(* Logix 5000 project; controller VET 1756-L62 rev 19.52; software revision 19.01; part 21 of 27 *)
(* tags used below, declared in another part *)
   _reset_locales : DINT;
   Batch : batch[10];
   Batch_buff : batch;
   Batch_Reportes : batch[100];
   comandos : DINT[10];
   db_input_cola : cola_almacenes;
   db_input_cola_batch_res : DINT;
   db_input_cola_flag : BOOL;
   dosificador : dosif_struct[20];
   Dosificar_LIQ_01 : PHASE;
   Dosificar_MAC_01 : PHASE;
   Dosificar_MAN_01 : PHASE;
   Dosificar_MIC_01 : PHASE;
   Dosificar_MIC_02 : PHASE;
   Dosificar_MID_01 : PHASE;
   hora_plc : DINT;
(* Interfaz_Equipment_Phase, continued *)

ROUTINE Dosificar_MIC_02   (* ladder *)
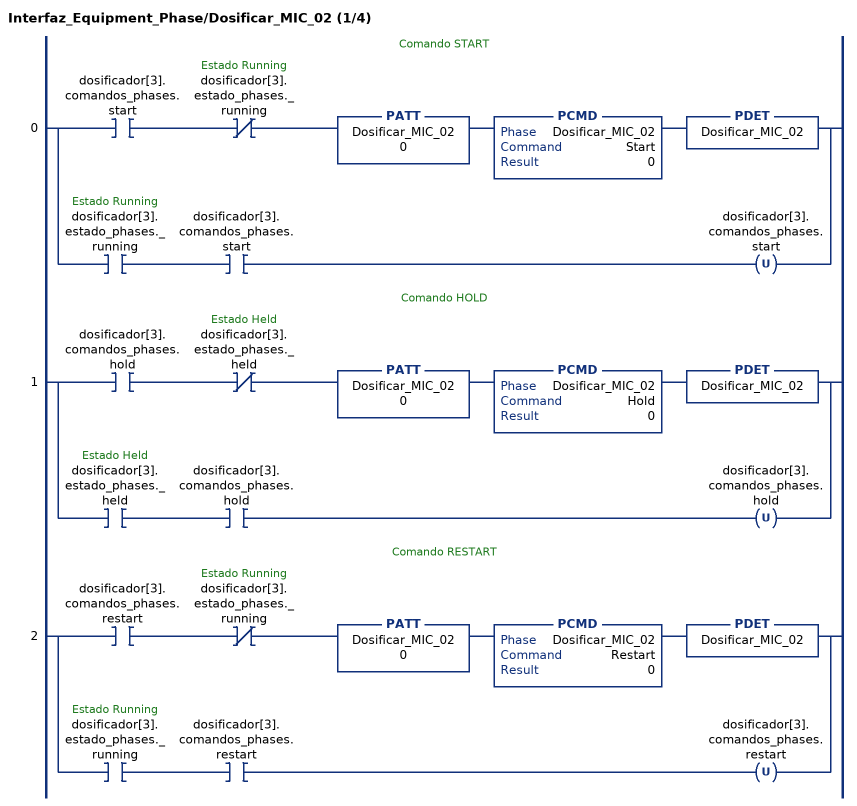
   // Comando START
   0: [XIC(dosificador[3].comandos_phases.start) XIO(dosificador[3].estado_phases._running) PATT(Dosificar_MIC_02,0) PCMD(Dosificar_MIC_02,Start,0) PDET(Dosificar_MIC_02) ,XIC(dosificador[3].estado_phases._running) XIC(dosificador[3].comandos_phases.start) OTU(dosificador[3].comandos_phases.start) ];
   // Comando HOLD
   1: [XIC(dosificador[3].comandos_phases.hold) XIO(dosificador[3].estado_phases._held) PATT(Dosificar_MIC_02,0) PCMD(Dosificar_MIC_02,Hold,0) PDET(Dosificar_MIC_02) ,XIC(dosificador[3].estado_phases._held) XIC(dosificador[3].comandos_phases.hold) OTU(dosificador[3].comandos_phases.hold) ];
   // Comando RESTART
   2: [XIC(dosificador[3].comandos_phases.restart) XIO(dosificador[3].estado_phases._running) PATT(Dosificar_MIC_02,0) PCMD(Dosificar_MIC_02,Restart,0) PDET(Dosificar_MIC_02) ,XIC(dosificador[3].estado_phases._running) XIC(dosificador[3].comandos_phases.restart) OTU(dosificador[3].comandos_phases.restart) ];
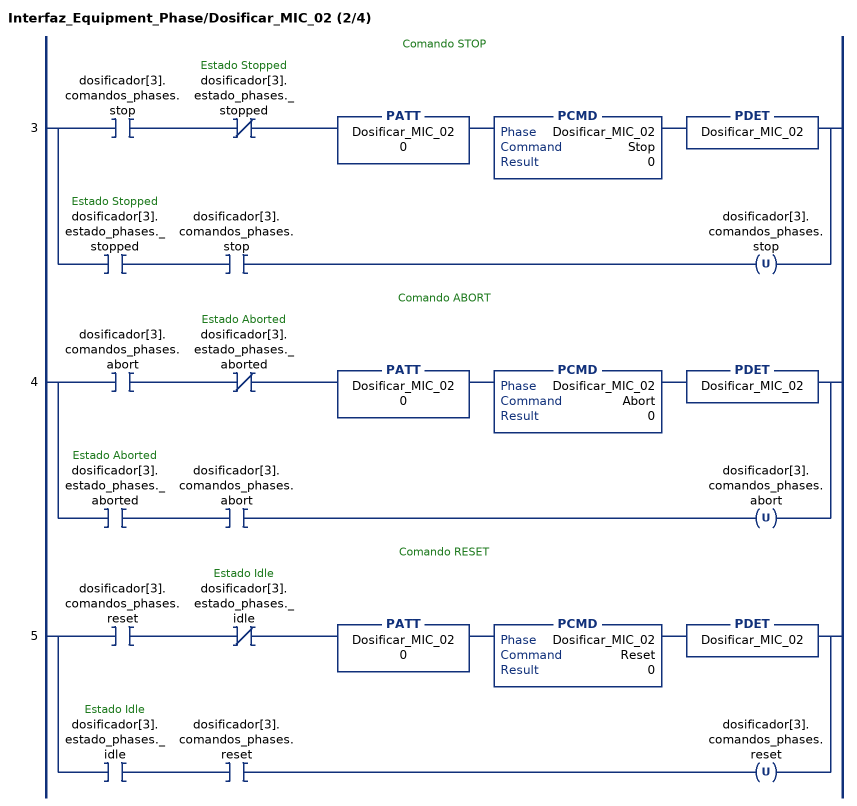
   // Comando STOP
   3: [XIC(dosificador[3].comandos_phases.stop) XIO(dosificador[3].estado_phases._stopped) PATT(Dosificar_MIC_02,0) PCMD(Dosificar_MIC_02,Stop,0) PDET(Dosificar_MIC_02) ,XIC(dosificador[3].estado_phases._stopped) XIC(dosificador[3].comandos_phases.stop) OTU(dosificador[3].comandos_phases.stop) ];
   // Comando ABORT
   4: [XIC(dosificador[3].comandos_phases.abort) XIO(dosificador[3].estado_phases._aborted) PATT(Dosificar_MIC_02,0) PCMD(Dosificar_MIC_02,Abort,0) PDET(Dosificar_MIC_02) ,XIC(dosificador[3].estado_phases._aborted) XIC(dosificador[3].comandos_phases.abort) OTU(dosificador[3].comandos_phases.abort) ];
   // Comando RESET
   5: [XIC(dosificador[3].comandos_phases.reset) XIO(dosificador[3].estado_phases._idle) PATT(Dosificar_MIC_02,0) PCMD(Dosificar_MIC_02,Reset,0) PDET(Dosificar_MIC_02) ,XIC(dosificador[3].estado_phases._idle) XIC(dosificador[3].comandos_phases.reset) OTU(dosificador[3].comandos_phases.reset) ];
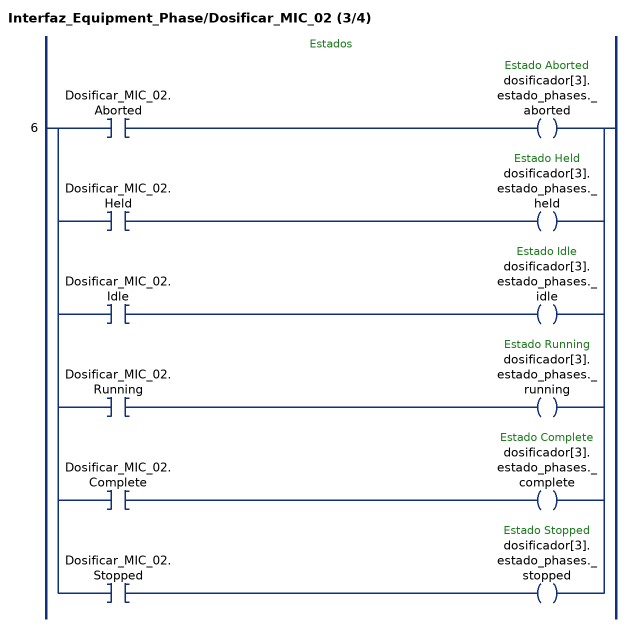
   // Estados
   6: [XIC(Dosificar_MIC_02.Aborted) OTE(dosificador[3].estado_phases._aborted) ,XIC(Dosificar_MIC_02.Held) OTE(dosificador[3].estado_phases._held) ,XIC(Dosificar_MIC_02.Idle) OTE(dosificador[3].estado_phases._idle) ,XIC(Dosificar_MIC_02.Running) OTE(dosificador[3].estado_phases._running) ,XIC(Dosificar_MIC_02.Complete) OTE(dosificador[3].estado_phases._complete) ,XIC(Dosificar_MIC_02.Stopped) OTE(dosificador[3].estado_phases._stopped) ];
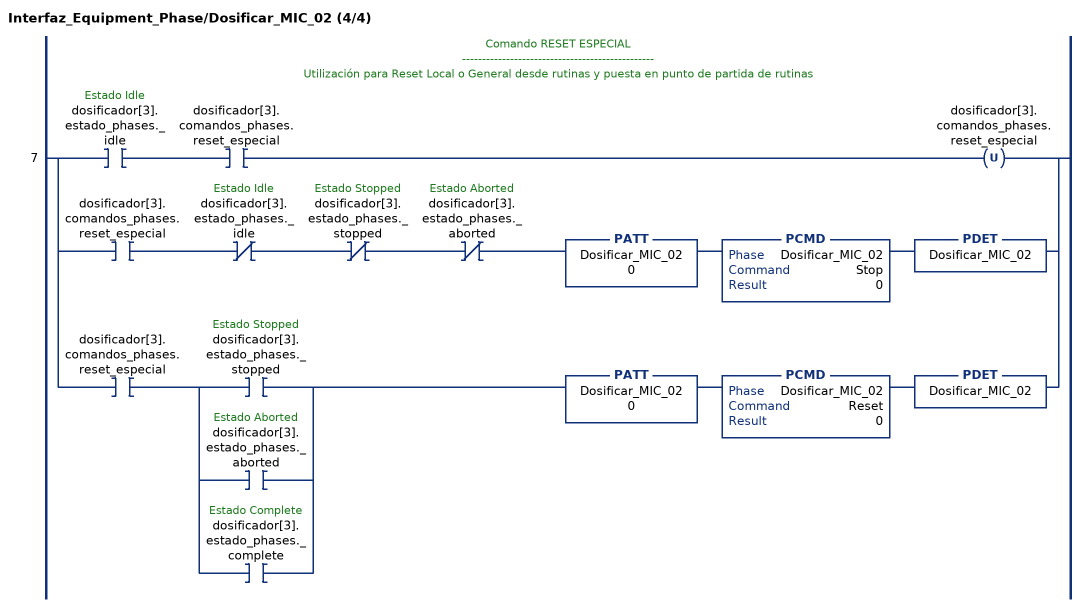
   // Comando RESET ESPECIAL
   // ------------------------------------------------
   // Utilización para Reset Local o General desde rutinas y puesta en punto de partida de rutinas
   7: [XIC(dosificador[3].estado_phases._idle) XIC(dosificador[3].comandos_phases.reset_especial) OTU(dosificador[3].comandos_phases.reset_especial) ,XIC(dosificador[3].comandos_phases.reset_especial) XIO(dosificador[3].estado_phases._idle) XIO(dosificador[3].estado_phases._stopped) XIO(dosificador[3].estado_phases._aborted) PATT(Dosificar_MIC_02,0) PCMD(Dosificar_MIC_02,Stop,0) PDET(Dosificar_MIC_02) ,XIC(dosificador[3].comandos_phases.reset_especial) [XIC(dosificador[3].estado_phases._stopped) ,XIC(dosificador[3].estado_phases._aborted) ,XIC(dosificador[3].estado_phases._complete) ] PATT(Dosificar_MIC_02,0) PCMD(Dosificar_MIC_02,Reset,0) PDET(Dosificar_MIC_02) ];
END_ROUTINE

ROUTINE Dosificar_MID_01   (* ladder *)
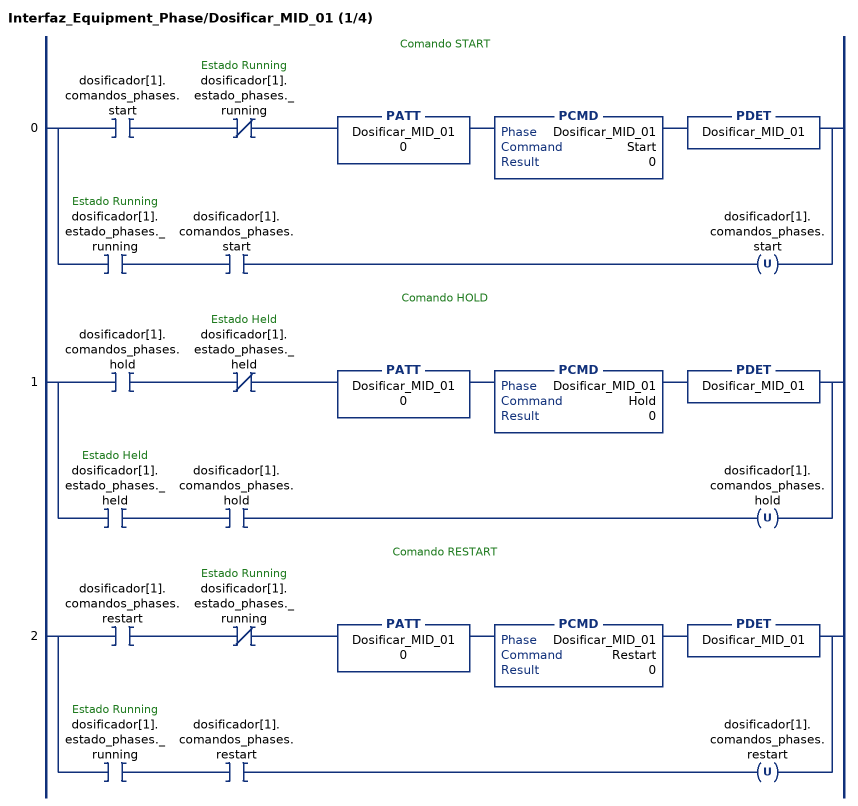
   // Comando START
   0: [XIC(dosificador[1].comandos_phases.start) XIO(dosificador[1].estado_phases._running) PATT(Dosificar_MID_01,0) PCMD(Dosificar_MID_01,Start,0) PDET(Dosificar_MID_01) ,XIC(dosificador[1].estado_phases._running) XIC(dosificador[1].comandos_phases.start) OTU(dosificador[1].comandos_phases.start) ];
   // Comando HOLD
   1: [XIC(dosificador[1].comandos_phases.hold) XIO(dosificador[1].estado_phases._held) PATT(Dosificar_MID_01,0) PCMD(Dosificar_MID_01,Hold,0) PDET(Dosificar_MID_01) ,XIC(dosificador[1].estado_phases._held) XIC(dosificador[1].comandos_phases.hold) OTU(dosificador[1].comandos_phases.hold) ];
   // Comando RESTART
   2: [XIC(dosificador[1].comandos_phases.restart) XIO(dosificador[1].estado_phases._running) PATT(Dosificar_MID_01,0) PCMD(Dosificar_MID_01,Restart,0) PDET(Dosificar_MID_01) ,XIC(dosificador[1].estado_phases._running) XIC(dosificador[1].comandos_phases.restart) OTU(dosificador[1].comandos_phases.restart) ];
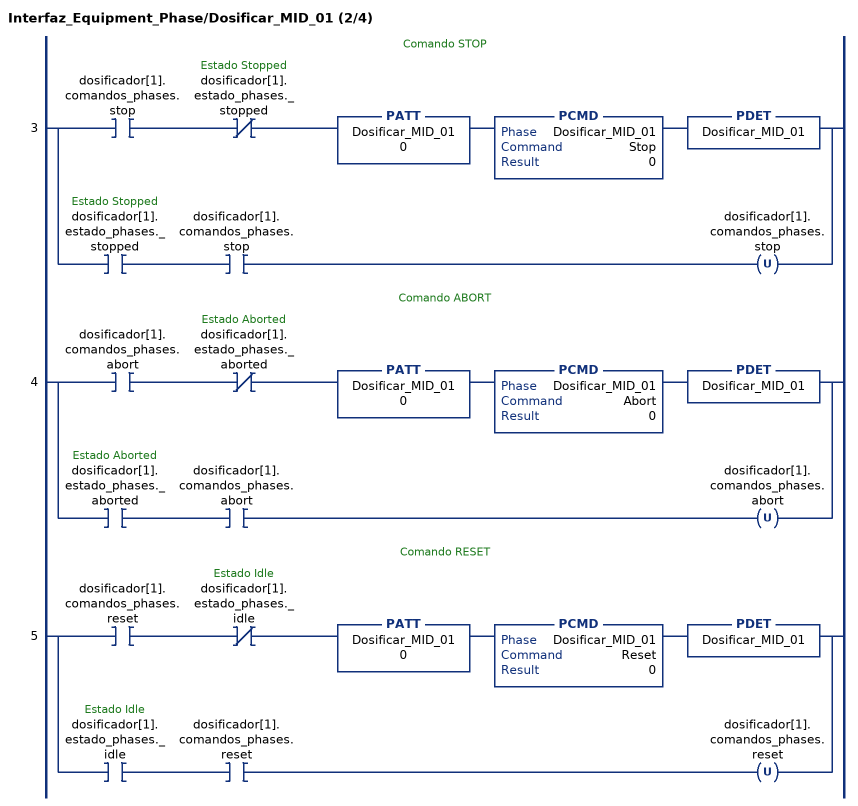
   // Comando STOP
   3: [XIC(dosificador[1].comandos_phases.stop) XIO(dosificador[1].estado_phases._stopped) PATT(Dosificar_MID_01,0) PCMD(Dosificar_MID_01,Stop,0) PDET(Dosificar_MID_01) ,XIC(dosificador[1].estado_phases._stopped) XIC(dosificador[1].comandos_phases.stop) OTU(dosificador[1].comandos_phases.stop) ];
   // Comando ABORT
   4: [XIC(dosificador[1].comandos_phases.abort) XIO(dosificador[1].estado_phases._aborted) PATT(Dosificar_MID_01,0) PCMD(Dosificar_MID_01,Abort,0) PDET(Dosificar_MID_01) ,XIC(dosificador[1].estado_phases._aborted) XIC(dosificador[1].comandos_phases.abort) OTU(dosificador[1].comandos_phases.abort) ];
   // Comando RESET
   5: [XIC(dosificador[1].comandos_phases.reset) XIO(dosificador[1].estado_phases._idle) PATT(Dosificar_MID_01,0) PCMD(Dosificar_MID_01,Reset,0) PDET(Dosificar_MID_01) ,XIC(dosificador[1].estado_phases._idle) XIC(dosificador[1].comandos_phases.reset) OTU(dosificador[1].comandos_phases.reset) ];
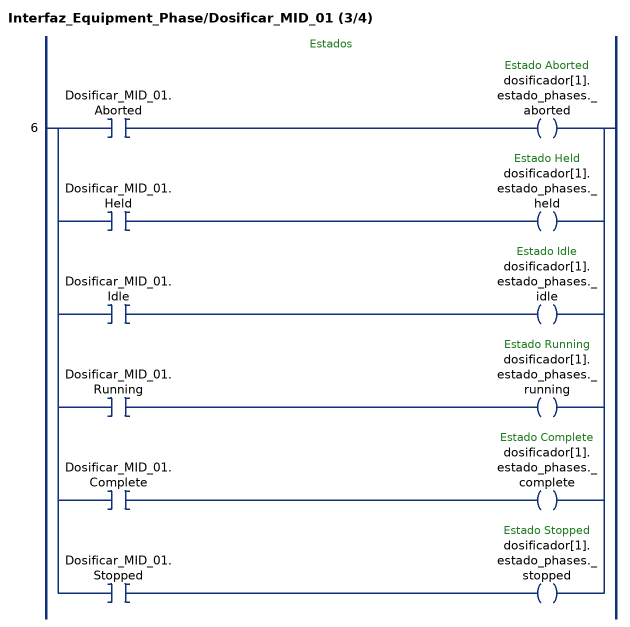
   // Estados
   6: [XIC(Dosificar_MID_01.Aborted) OTE(dosificador[1].estado_phases._aborted) ,XIC(Dosificar_MID_01.Held) OTE(dosificador[1].estado_phases._held) ,XIC(Dosificar_MID_01.Idle) OTE(dosificador[1].estado_phases._idle) ,XIC(Dosificar_MID_01.Running) OTE(dosificador[1].estado_phases._running) ,XIC(Dosificar_MID_01.Complete) OTE(dosificador[1].estado_phases._complete) ,XIC(Dosificar_MID_01.Stopped) OTE(dosificador[1].estado_phases._stopped) ];
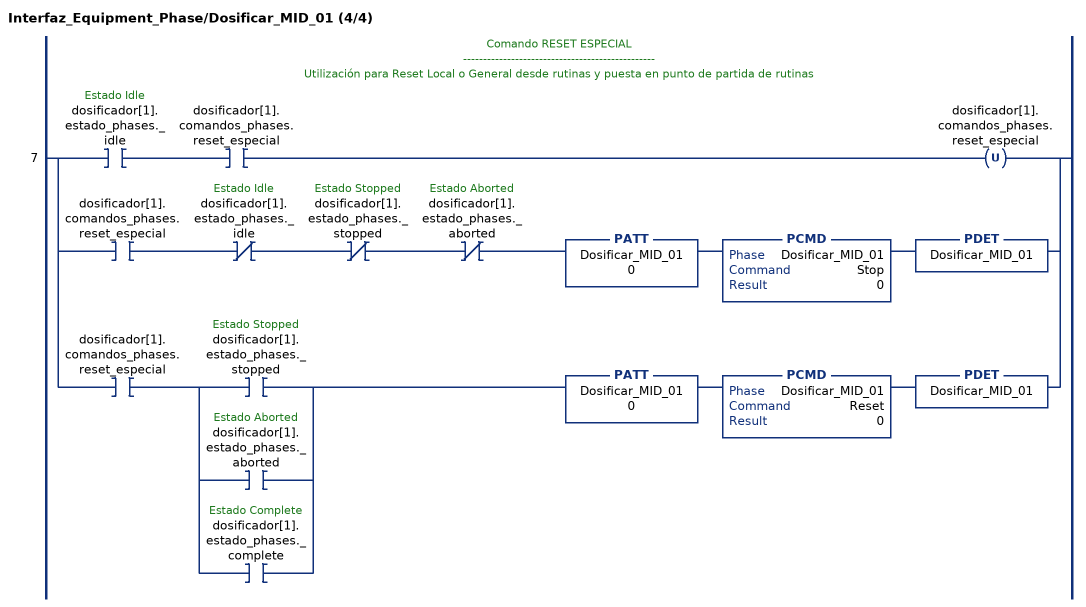
   // Comando RESET ESPECIAL
   // ------------------------------------------------
   // Utilización para Reset Local o General desde rutinas y puesta en punto de partida de rutinas
   7: [XIC(dosificador[1].estado_phases._idle) XIC(dosificador[1].comandos_phases.reset_especial) OTU(dosificador[1].comandos_phases.reset_especial) ,XIC(dosificador[1].comandos_phases.reset_especial) XIO(dosificador[1].estado_phases._idle) XIO(dosificador[1].estado_phases._stopped) XIO(dosificador[1].estado_phases._aborted) PATT(Dosificar_MID_01,0) PCMD(Dosificar_MID_01,Stop,0) PDET(Dosificar_MID_01) ,XIC(dosificador[1].comandos_phases.reset_especial) [XIC(dosificador[1].estado_phases._stopped) ,XIC(dosificador[1].estado_phases._aborted) ,XIC(dosificador[1].estado_phases._complete) ] PATT(Dosificar_MID_01,0) PCMD(Dosificar_MID_01,Reset,0) PDET(Dosificar_MID_01) ];
END_ROUTINE

ROUTINE main   (* ladder *)
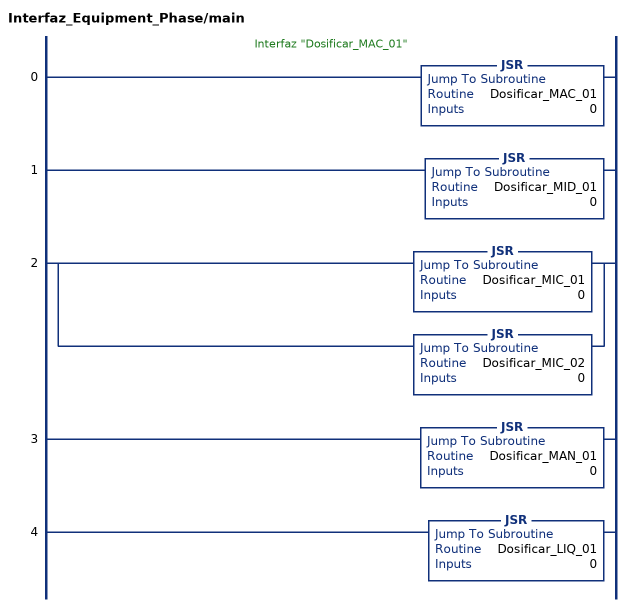
   // Interfaz "Dosificar_MAC_01"
   0: JSR(Dosificar_MAC_01,0);
   1: JSR(Dosificar_MID_01,0);
   2: [JSR(Dosificar_MIC_01,0) ,JSR(Dosificar_MIC_02,0) ];
   3: JSR(Dosificar_MAN_01,0);
   4: JSR(Dosificar_LIQ_01,0);
END_ROUTINE
END_PROGRAM

PROGRAM Main   (* main routine main *)
VAR
   _reset_local : ALIAS FOR _reset_locales.0;
   batch_in : batch := (Head.folio := 32, Head.orden := -3, Head.formula := 'DUMMY', Head.estado := 5, Head.correlativo := 2, Head.total_batch := 20, Head.peso_teorico := 1733.0, Data.codigo[0] := 81, Data.codigo[1] := 51, Data.codigo[2] := 53, Data.codigo[3] := 55, Data.codigo[4] := 57, Data.codigo[5] := 67, Data.codigo[6] := 68, Data.codigo[7] := 69, Data.codigo[8] := 70, Data.codigo[9] := 74, Data.codigo[10] := 75, Data.codigo[11] := 76, Data.codigo[12] := 77, Data.codigo[13] := 60, Data.codigo[14] := 62, Data.codigo[15] := 64, Data.codigo[16] := 66, Data.peso_f[0] := 70.0, Data.peso_f[1] := 400.0, Data.peso_f[2] := 350.0, Data.peso_f[3] := 175.0, Data.peso_f[4] := 225.0, Data.peso_f[5] := 30.0, Data.peso_f[6] := 25.0, Data.peso_f[7] := 17.5, Data.peso_f[8] := 17.5, Data.peso_f[9] := 30.0, Data.peso_f[10] := 5.0, Data.peso_f[11] := 4.0, Data.peso_f[12] := 4.0, Data.peso_f[13] := 125.0, Data.peso_f[14] := 125.0, Data.peso_f[15] := 65.0, Data.peso_f[16] := 65.0);
   batch_out : batch;
   db1_var_batch : variables_procedimientos := (trigger[0] := 1, trigger[1] := 1, trigger[2] := 1, trigger[3] := 1, handshake[0] := 1, handshake[1] := 1, handshake[2] := 1, in_tstamp[0] := 18273253, in_tstamp[1] := 18273653, in_tstamp[2] := 18274003, in_tstamp[3] := 11123107, out_tstamp[0] := 18273253, out_tstamp[2] := 18274003, D[0] := 3, D[1] := 32, T[0].PRE := 2000, T[1].PRE := 10000, T[2].PRE := 2000, T[3].PRE := 10000, T[4].PRE := 2000, T[5].PRE := 10000);
        .D[0].1   // Habilitación Recepción Automática
        .D[0].0   // Resumen Dehabilitación
        .D[0]   // Bits Estados
        .D[1]   // Folio - Pedir batch
   db2_cola_res : DINT[20] := ([0] := 32, [1] := 27862, [2] := 39951);
   db2_var_res : variables_procedimientos := (step_idx := 20, trigger[0] := 1, handshake[0] := -1, in_tstamp[0] := 18464153, D[0] := 32, i0 := 1, SetD[0] := 20, T[0].PRE := 3000, T[1].PRE := 10000, T[1].ACC := 4992, T[1].EN := 1, T[1].TT := 1);
   db3_var_rep : variables_procedimientos;
   db4_cola_mc : cola_almacenes[100] := ([0].origen := 31, [0].destino := 1000, [0].cantidad := 16.200012, [0].folio_op := 39951, [0].fecha := 20140306, [0].hora := 1163858, [1].origen := 31, [1].destino := 1000, [1].cantidad := 16.299988, [1].folio_op := 39973, [1].fecha := 20140306, [1].hora := 1170439, [2].origen := 71, [2].destino := 1000, [2].cantidad := 2.015625, [2].folio_op := 39973, [2].fecha := 20140306, [2].hora := 1170440, [3].origen := 31, [3].destino := 1000, [3].cantidad := 16.600006, [3].folio_op := 39975, [3].fecha := 20140306, [3].hora := 1172638, [4].origen := 70, [4].destino := 1000, [4].cantidad := 31.046875, [4].folio_op := 39889, [4].fecha := 20140306, [4].hora := 1174046, [5].origen := 31, [5].destino := 1000, [5].cantidad := 16.800018, [5].folio_op := 39977, [5].fecha := 20140306, [5].hora := 1175226, [6].origen := 32, [6].destino := 1000, [6].cantidad := 10.300018, [6].folio_op := 39977, [6].fecha := 20140306, [6].hora := 1175710, [7].origen := 70, [7].destino := 1000, [7].cantidad := 31.0, [7].folio_op := 39815, [7].fecha := 20140306, [7].hora := 1122359, [8].origen := 71, [8].destino := 1000, [8].cantidad := 2.0, [8].folio_op := 39937, [8].fecha := 20140306, [8].hora := 1124946, [9].origen := 31, [9].destino := 1000, [9].cantidad := 16.800018, [9].folio_op := 39937, [9].fecha := 20140306, [9].hora := 1124947,
        [10].origen := 19, [10].destino := 1000, [10].cantidad := 656.0, [10].folio_op := 39903, [10].fecha := 20140306, [10].hora := 1125834, [11].origen := 31, [11].destino := 1000, [11].cantidad := 16.299988, [11].folio_op := 39942, [11].fecha := 20140306, [11].hora := 1135834, [12].origen := 101, [12].destino := 1000, [12].cantidad := 50.4375, [12].folio_op := 39904, [12].fecha := 20140306, [12].hora := 1141004, [13].origen := 16, [13].destino := 25, [14].origen := 16, [14].destino := 25, [15].origen := 31, [15].destino := 1000, [15].cantidad := 16.5, [15].folio_op := 39945, [15].fecha := 20140306, [15].hora := 1151258, [16].origen := 31, [16].destino := 1000, [16].cantidad := 16.5, [16].folio_op := 39946, [16].fecha := 20140306, [16].hora := 1152347, [17].origen := 31, [17].destino := 1000, [17].cantidad := 16.799988, [17].folio_op := 39947, [17].fecha := 20140306, [17].hora := 1153707, [18].origen := 31, [18].destino := 1000, [18].cantidad := 16.200012, [18].folio_op := 39948, [18].fecha := 20140306, [18].hora := 1160218, [19].origen := 31, [19].destino := 1000, [19].cantidad := 16.800003, [19].folio_op := 39949, [19].fecha := 20140306, [19].hora := 1161219);
   db4_var_mc : variables_procedimientos;
   db5_var_rep : variables_procedimientos := (i0 := 50, i1 := 50, SetD[0] := 100);
        .I0   // Largo Actual Cola
        .SETD[0]   // Largo Maximo Cola
        .I1   // Próximo a la Cola
        .I2   // Primero en Cola
   var_wd : variables_procedimientos := (step_idx := 10, in_tstamp[0] := 18464753, T[0].PRE := 20000, T[0].ACC := 1992, T[0].EN := 1, T[0].TT := 1, T[1].PRE := 10000);
   watchdog : BOOL;
END_VAR

ROUTINE aux_manejo_cola   (* ladder *)
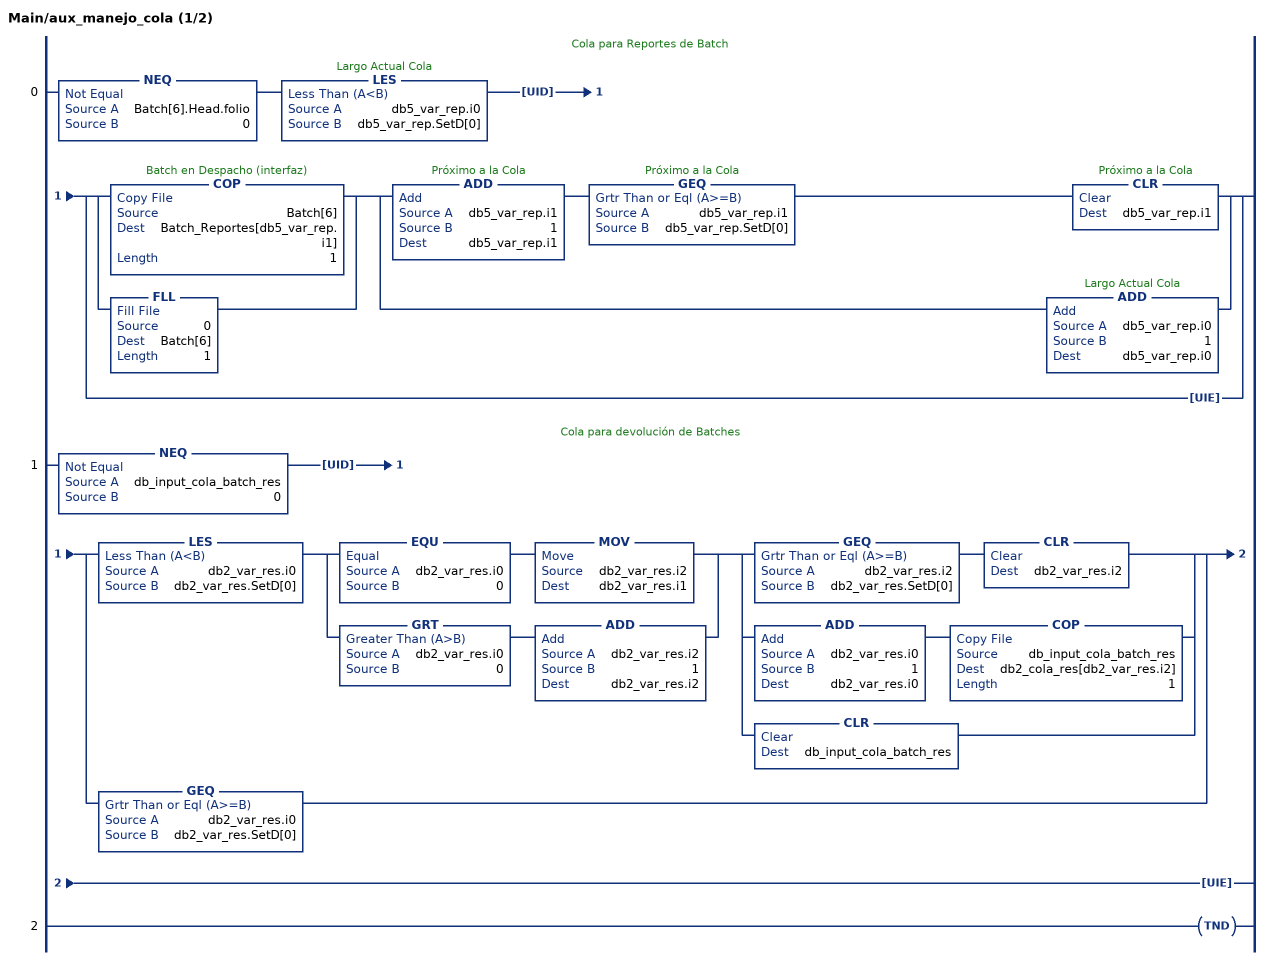
   // Cola para Reportes de Batch
   0: NEQ(Batch[6].Head.folio,0)LES(db5_var_rep.i0,db5_var_rep.SetD[0])UID()[[COP(Batch[6],Batch_Reportes[db5_var_rep.i1],1) ,FLL(0,Batch[6],1) ] [ADD(db5_var_rep.i1,1,db5_var_rep.i1) GEQ(db5_var_rep.i1,db5_var_rep.SetD[0]) CLR(db5_var_rep.i1) ,ADD(db5_var_rep.i0,1,db5_var_rep.i0) ] ,UIE() ];
   // Cola para devolución de Batches
   1: NEQ(db_input_cola_batch_res,0)UID()[LES(db2_var_res.i0,db2_var_res.SetD[0]) [EQU(db2_var_res.i0,0) MOV(db2_var_res.i2,db2_var_res.i1) ,GRT(db2_var_res.i0,0) ADD(db2_var_res.i2,1,db2_var_res.i2) ] [GEQ(db2_var_res.i2,db2_var_res.SetD[0]) CLR(db2_var_res.i2) ,ADD(db2_var_res.i0,1,db2_var_res.i0) COP(db_input_cola_batch_res,db2_cola_res[db2_var_res.i2],1) ,CLR(db_input_cola_batch_res) ] ,GEQ(db2_var_res.i0,db2_var_res.SetD[0]) ]UIE();
   2: TND();
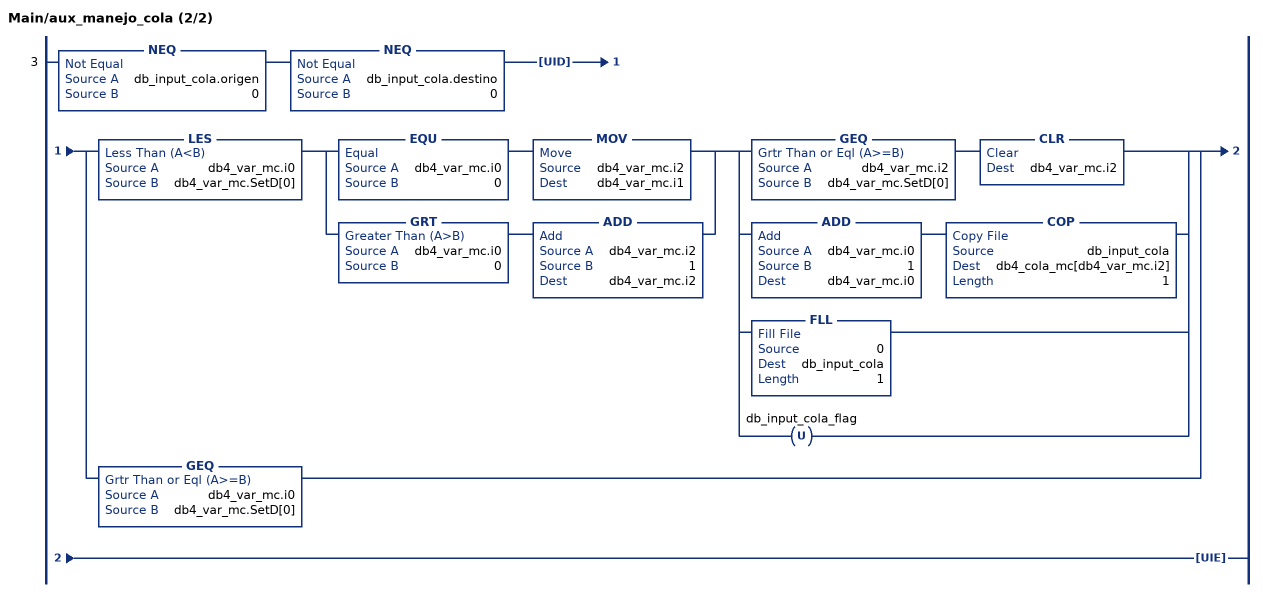
   3: NEQ(db_input_cola.origen,0)NEQ(db_input_cola.destino,0)UID()[LES(db4_var_mc.i0,db4_var_mc.SetD[0]) [EQU(db4_var_mc.i0,0) MOV(db4_var_mc.i2,db4_var_mc.i1) ,GRT(db4_var_mc.i0,0) ADD(db4_var_mc.i2,1,db4_var_mc.i2) ] [GEQ(db4_var_mc.i2,db4_var_mc.SetD[0]) CLR(db4_var_mc.i2) ,ADD(db4_var_mc.i0,1,db4_var_mc.i0) COP(db_input_cola,db4_cola_mc[db4_var_mc.i2],1) ,FLL(0,db_input_cola,1) ,OTU(db_input_cola_flag) ] ,GEQ(db4_var_mc.i0,db4_var_mc.SetD[0]) ]UIE();
END_ROUTINE

ROUTINE db0_watchdog   (* ladder *)
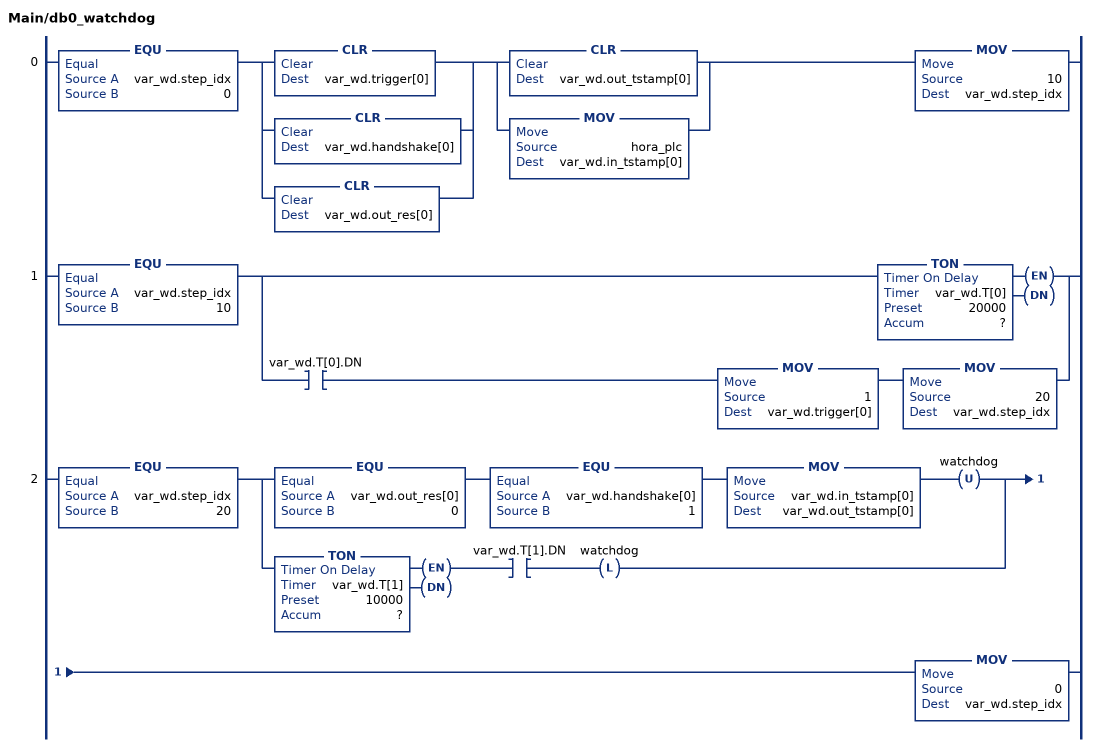
   0: EQU(var_wd.step_idx,0)[CLR(var_wd.trigger[0]) ,CLR(var_wd.handshake[0]) ,CLR(var_wd.out_res[0]) ][CLR(var_wd.out_tstamp[0]) ,MOV(hora_plc,var_wd.in_tstamp[0]) ]MOV(10,var_wd.step_idx);
   1: EQU(var_wd.step_idx,10)[TON(var_wd.T[0],?,?) ,XIC(var_wd.T[0].DN) MOV(1,var_wd.trigger[0]) MOV(20,var_wd.step_idx) ];
   2: EQU(var_wd.step_idx,20)[EQU(var_wd.out_res[0],0) EQU(var_wd.handshake[0],1) MOV(var_wd.in_tstamp[0],var_wd.out_tstamp[0]) OTU(watchdog) ,TON(var_wd.T[1],?,?) XIC(var_wd.T[1].DN) OTL(watchdog) ]MOV(0,var_wd.step_idx);
END_ROUTINE

ROUTINE db1_obtener_batch   (* ladder *)
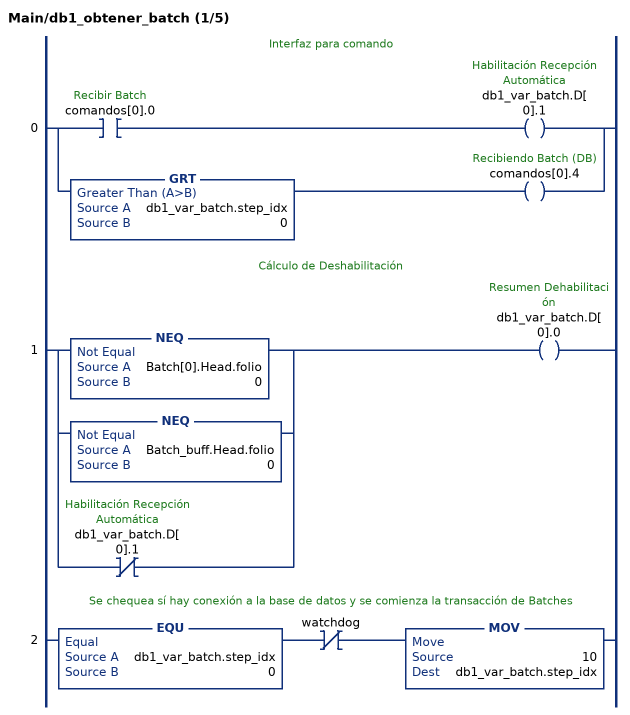
   // Interfaz para comando
   0: [XIC(comandos[0].0) OTE(db1_var_batch.D[0].1) ,GRT(db1_var_batch.step_idx,0) OTE(comandos[0].4) ];
   // Cálculo de Deshabilitación
   1: [NEQ(Batch[0].Head.folio,0) ,NEQ(Batch_buff.Head.folio,0) ,XIO(db1_var_batch.D[0].1) ]OTE(db1_var_batch.D[0].0);
   // Se chequea sí hay conexión a la base de datos y se comienza la transacción de Batches
   2: EQU(db1_var_batch.step_idx,0)XIO(watchdog)MOV(10,db1_var_batch.step_idx);
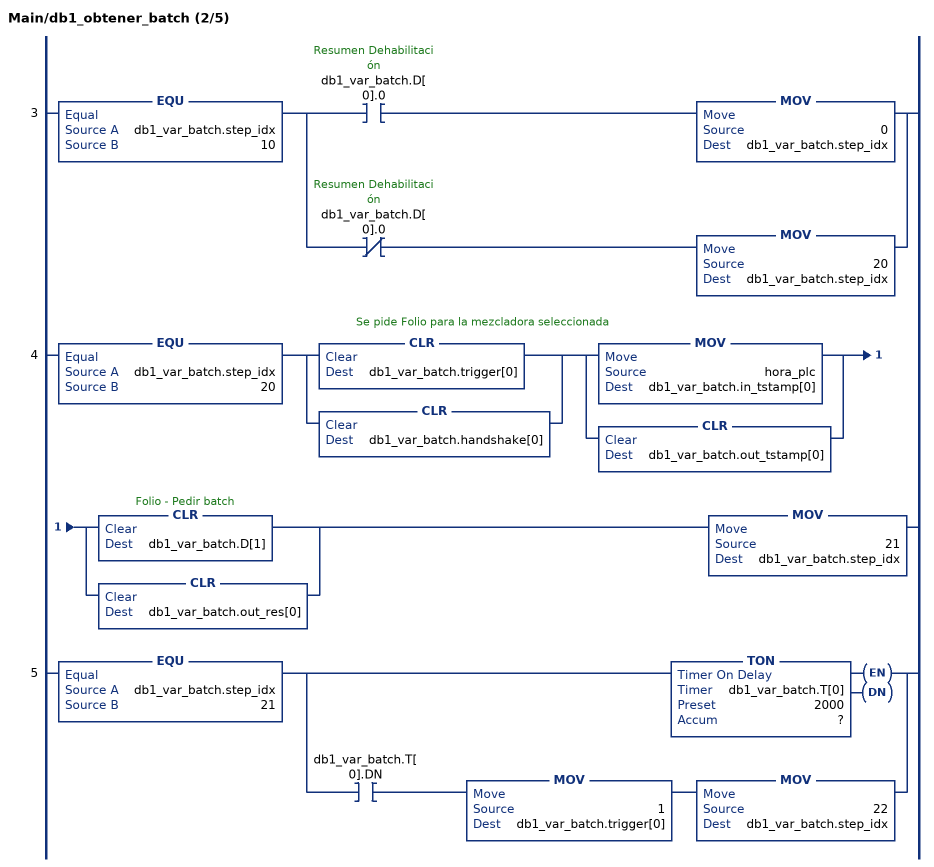
   3: EQU(db1_var_batch.step_idx,10)[XIC(db1_var_batch.D[0].0) MOV(0,db1_var_batch.step_idx) ,XIO(db1_var_batch.D[0].0) MOV(20,db1_var_batch.step_idx) ];
   // Se pide Folio para la mezcladora seleccionada
   4: EQU(db1_var_batch.step_idx,20)[CLR(db1_var_batch.trigger[0]) ,CLR(db1_var_batch.handshake[0]) ][MOV(hora_plc,db1_var_batch.in_tstamp[0]) ,CLR(db1_var_batch.out_tstamp[0]) ][CLR(db1_var_batch.D[1]) ,CLR(db1_var_batch.out_res[0]) ]MOV(21,db1_var_batch.step_idx);
   5: EQU(db1_var_batch.step_idx,21)[TON(db1_var_batch.T[0],?,?) ,XIC(db1_var_batch.T[0].DN) MOV(1,db1_var_batch.trigger[0]) MOV(22,db1_var_batch.step_idx) ];
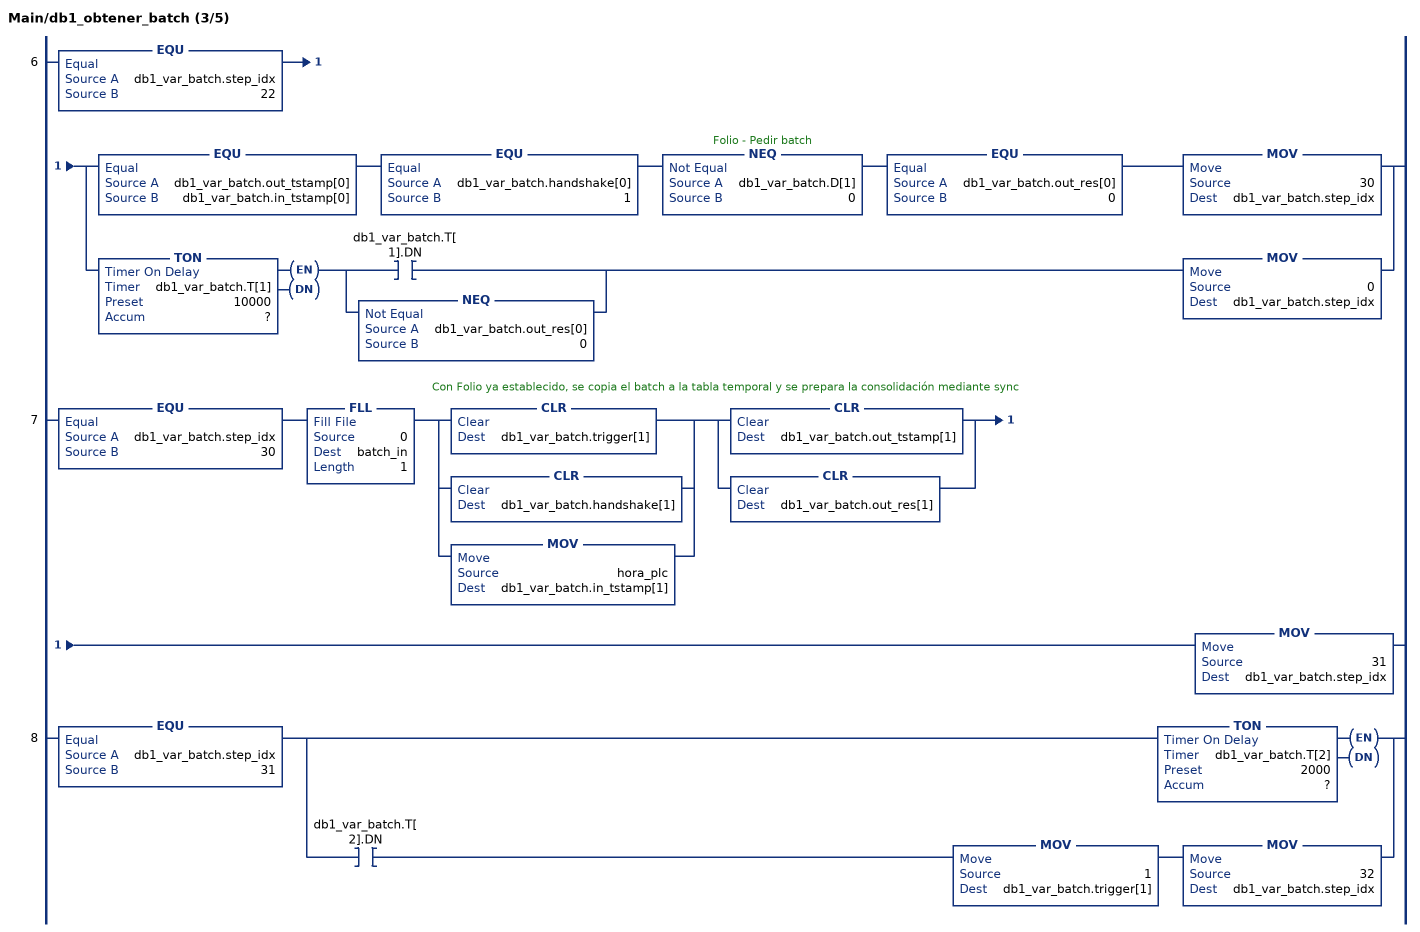
   6: EQU(db1_var_batch.step_idx,22)[EQU(db1_var_batch.out_tstamp[0],db1_var_batch.in_tstamp[0]) EQU(db1_var_batch.handshake[0],1) NEQ(db1_var_batch.D[1],0) EQU(db1_var_batch.out_res[0],0) MOV(30,db1_var_batch.step_idx) ,TON(db1_var_batch.T[1],?,?) [XIC(db1_var_batch.T[1].DN) ,NEQ(db1_var_batch.out_res[0],0) ] MOV(0,db1_var_batch.step_idx) ];
   // Con Folio ya establecido, se copia el batch a la tabla temporal y se prepara la consolidación mediante sync
   7: EQU(db1_var_batch.step_idx,30)FLL(0,batch_in,1)[CLR(db1_var_batch.trigger[1]) ,CLR(db1_var_batch.handshake[1]) ,MOV(hora_plc,db1_var_batch.in_tstamp[1]) ][CLR(db1_var_batch.out_tstamp[1]) ,CLR(db1_var_batch.out_res[1]) ]MOV(31,db1_var_batch.step_idx);
   8: EQU(db1_var_batch.step_idx,31)[TON(db1_var_batch.T[2],?,?) ,XIC(db1_var_batch.T[2].DN) MOV(1,db1_var_batch.trigger[1]) MOV(32,db1_var_batch.step_idx) ];
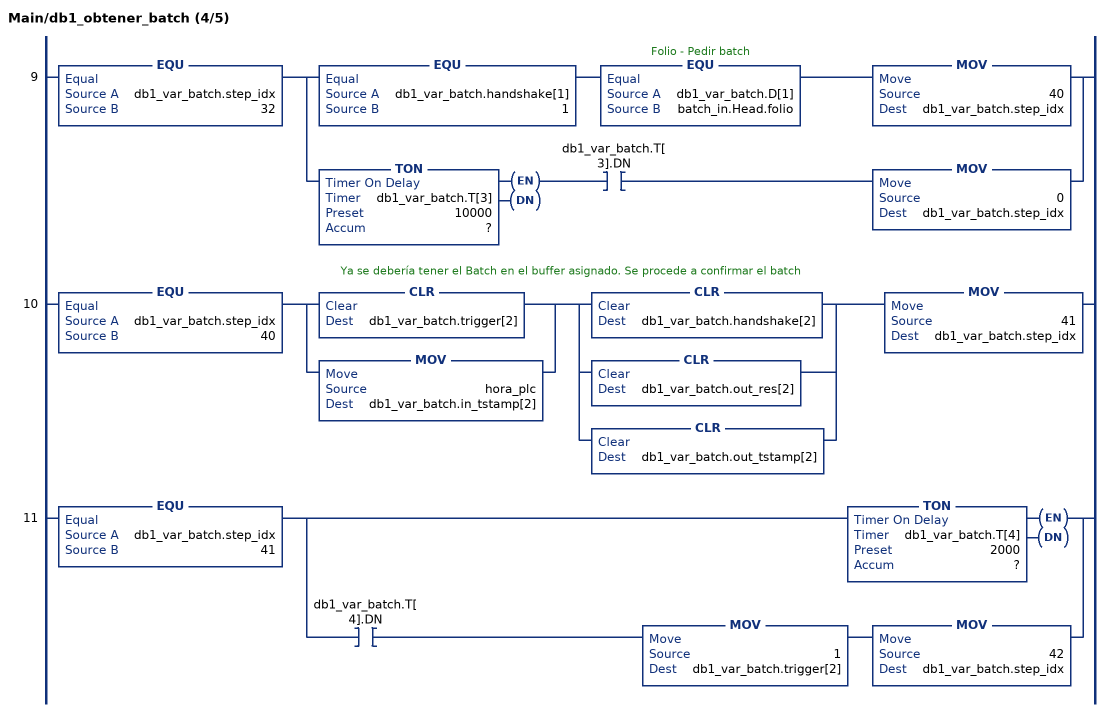
   9: EQU(db1_var_batch.step_idx,32)[EQU(db1_var_batch.handshake[1],1) EQU(db1_var_batch.D[1],batch_in.Head.folio) MOV(40,db1_var_batch.step_idx) ,TON(db1_var_batch.T[3],?,?) XIC(db1_var_batch.T[3].DN) MOV(0,db1_var_batch.step_idx) ];
   // Ya se debería tener el Batch en el buffer asignado. Se procede a confirmar el batch
   10: EQU(db1_var_batch.step_idx,40)[CLR(db1_var_batch.trigger[2]) ,MOV(hora_plc,db1_var_batch.in_tstamp[2]) ][CLR(db1_var_batch.handshake[2]) ,CLR(db1_var_batch.out_res[2]) ,CLR(db1_var_batch.out_tstamp[2]) ]MOV(41,db1_var_batch.step_idx);
   11: EQU(db1_var_batch.step_idx,41)[TON(db1_var_batch.T[4],?,?) ,XIC(db1_var_batch.T[4].DN) MOV(1,db1_var_batch.trigger[2]) MOV(42,db1_var_batch.step_idx) ];
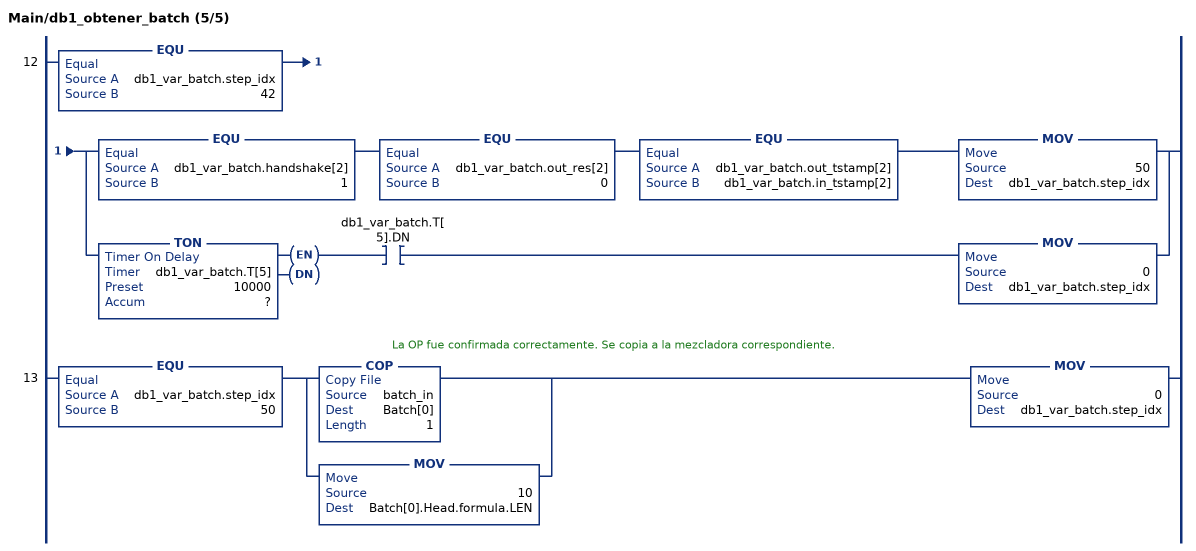
   12: EQU(db1_var_batch.step_idx,42)[EQU(db1_var_batch.handshake[2],1) EQU(db1_var_batch.out_res[2],0) EQU(db1_var_batch.out_tstamp[2],db1_var_batch.in_tstamp[2]) MOV(50,db1_var_batch.step_idx) ,TON(db1_var_batch.T[5],?,?) XIC(db1_var_batch.T[5].DN) MOV(0,db1_var_batch.step_idx) ];
   // La OP fue confirmada correctamente. Se copia a la mezcladora correspondiente.
   13: EQU(db1_var_batch.step_idx,50)[COP(batch_in,Batch[0],1) ,MOV(10,Batch[0].Head.formula.LEN) ]MOV(0,db1_var_batch.step_idx);
END_ROUTINE

ROUTINE db2_devolver_op   (* ladder *)
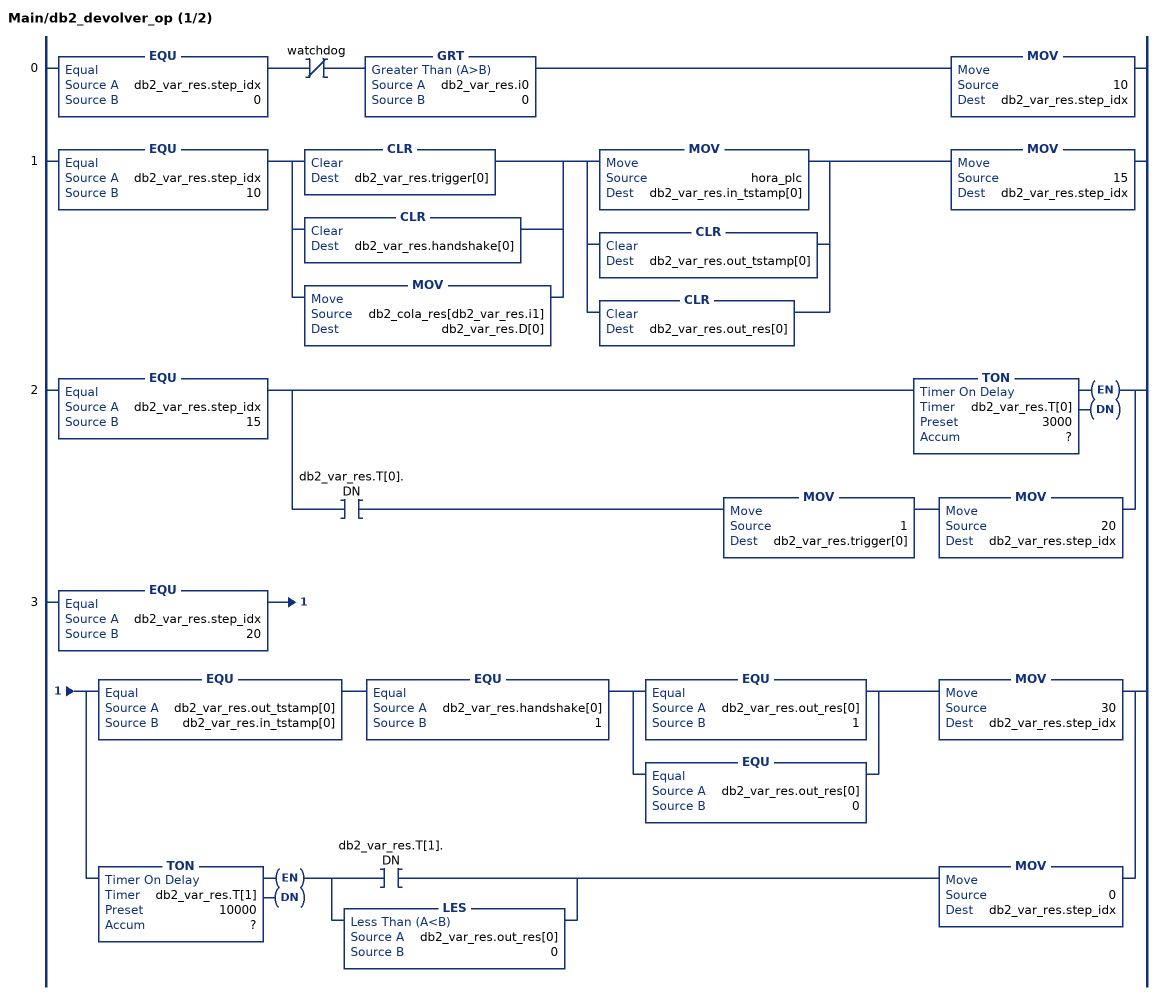
   0: EQU(db2_var_res.step_idx,0)XIO(watchdog)GRT(db2_var_res.i0,0)MOV(10,db2_var_res.step_idx);
   1: EQU(db2_var_res.step_idx,10)[CLR(db2_var_res.trigger[0]) ,CLR(db2_var_res.handshake[0]) ,MOV(db2_cola_res[db2_var_res.i1],db2_var_res.D[0]) ][MOV(hora_plc,db2_var_res.in_tstamp[0]) ,CLR(db2_var_res.out_tstamp[0]) ,CLR(db2_var_res.out_res[0]) ]MOV(15,db2_var_res.step_idx);
   2: EQU(db2_var_res.step_idx,15)[TON(db2_var_res.T[0],?,?) ,XIC(db2_var_res.T[0].DN) MOV(1,db2_var_res.trigger[0]) MOV(20,db2_var_res.step_idx) ];
   3: EQU(db2_var_res.step_idx,20)[EQU(db2_var_res.out_tstamp[0],db2_var_res.in_tstamp[0]) EQU(db2_var_res.handshake[0],1) [EQU(db2_var_res.out_res[0],1) ,EQU(db2_var_res.out_res[0],0) ] MOV(30,db2_var_res.step_idx) ,TON(db2_var_res.T[1],?,?) [XIC(db2_var_res.T[1].DN) ,LES(db2_var_res.out_res[0],0) ] MOV(0,db2_var_res.step_idx) ];
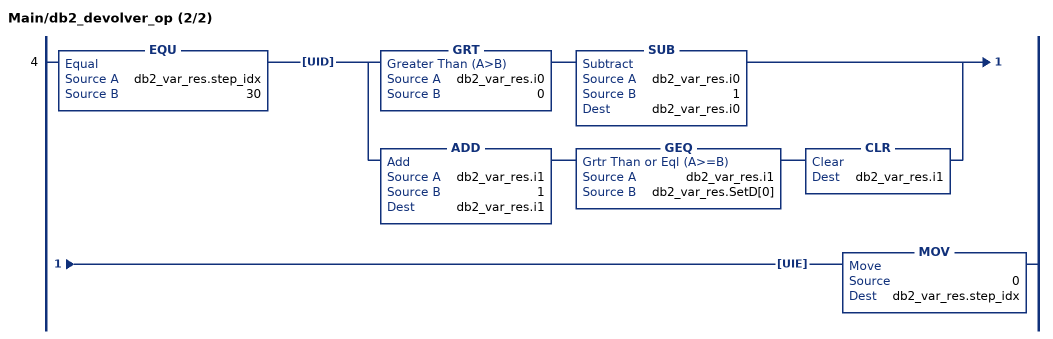
   4: EQU(db2_var_res.step_idx,30)UID()[GRT(db2_var_res.i0,0) SUB(db2_var_res.i0,1,db2_var_res.i0) ,ADD(db2_var_res.i1,1,db2_var_res.i1) GEQ(db2_var_res.i1,db2_var_res.SetD[0]) CLR(db2_var_res.i1) ]UIE()MOV(0,db2_var_res.step_idx);
END_ROUTINE
